Fanuc KAREL source: kc00014.KL

-- PROVISIONAL review KL for V1013-1; original PC SHA256 cf781308298e23838a29dbd06ac31929fb6ade658a39d2c9195836cc74c15825
-- Incomplete behavior may be omitted. Consult companion uncertainty JSON. Do not deploy.
PROGRAM KC00014
%NOLOCKGROUP
BEGIN
  -- UNRESOLVED_PC offsets 5-15; opcodes 27,31,23
  -- UNRESOLVED_PC offsets 20-24; opcodes 7F
END KC00014
